TEXTLIST Breaker_Status
  0 = 'HEALTHY'
  1 = 'FAULT'
   = ''
END_TEXTLIST

(* stored: Version 1.1.0.1, ProductVersion 3.1.4024.12
   TextList Breaker_Status: Id {ac26fe50-44b4-4940-bed2-9dac4967c633} *)
